// TIA Portal V19 export
VAR_GLOBAL   // PLC tag table "DemoCase"
   POT1_Upper_1500 AT %IW6 : Int;   // connected to AI channel 2
   TopLights_red_1500 AT %Q10.1 : Bool;   // TopLight red 1=on 0=off
   TopLights_green_1500 AT %Q10.0 : Bool;   // TopLight green 1=on 0=off
   POT2_Lower_1500 AT %IW14 : Int;   // connected to AI channel 6
   TopLights_blue_1500 AT %Q10.2 : Bool;   // TopLight blue 1=on 0=off
   PB_Green_1500 AT %I0.0 : Bool;
   PB_Blue_1500 AT %I0.1 : Bool;
   PB_Green_Lamp AT %Q8.0 : Bool;
   PB_Blue_Lamp AT %Q8.1 : Bool;
   POT4_G120 AT %MD30 : Real;
   HMI_IO_Test AT %M10.4 : Bool;
   PB_Green_1200 AT %M60.0 : Bool;
   PB_Blue_1200 AT %M60.1 : Bool;
   POT3_Upper_1200 AT %MW62 : Int;
   PB_Green_Lamp_1200 AT %M64.0 : Bool;
   PB_Blue_Lamp_1200 AT %M64.1 : Bool;
   TopLights_Green_1200 AT %M64.5 : Bool;
   TopLights_Red_1200 AT %M64.6 : Bool;
   TopLights_Blue_1200 AT %M64.7 : Bool;
   "1200_Inputs" AT %MB60 : Byte;
   "1200_Outputs" AT %MB64 : Byte;
   "1200_All_Inputs" AT %MD60 : DWord;
   OS6 AT %M11.4 : Bool;
   "Out to 1200" AT %QW100 : Int;
   "Red Latch" AT %M11.5 : Bool;
   "Green Latch" AT %M11.6 : Bool;
   GateClosed AT %M11.7 : Bool;
   "Blue Latch" AT %M20.3 : Bool;
   Coordination AT %MW36 : Int;
END_VAR
